// SIMATIC S7-200 project (STEP 7-Micro/WIN), CPU 224XP REL 02.01

SYMBOL_TABLE USUARIO1
S1_VERDE         Q0.0
S1_AMBAR         Q0.1
S1_ROJO          Q0.2
S2_VERDE         Q0.3
S2_AMBAR         Q0.4
S2_ROJO          Q0.5
END_SYMBOL_TABLE

SYMBOL_TABLE Símbolos S7-200
Primer_ciclo_ON  SM0.1    // ON sólo en el primer ciclo
END_SYMBOL_TABLE

ORGANIZATION_BLOCK PRINCIPAL:OB1
TITLE=COMENTARIOS DEL PROGRAMA
BEGIN
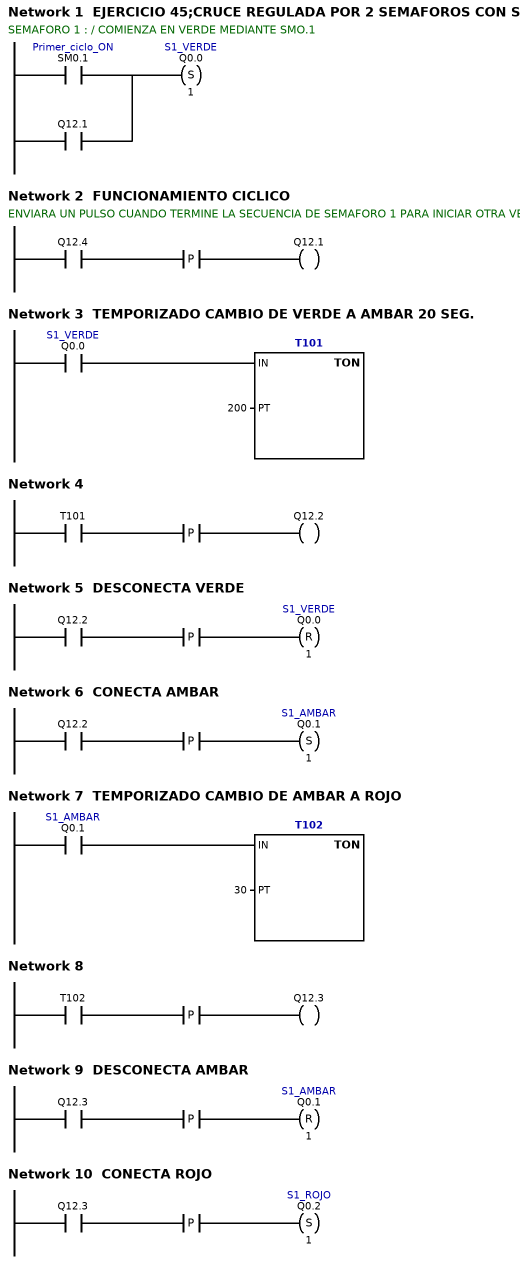
Network 1 // EJERCICIO 45;CRUCE REGULADA POR 2 SEMAFOROS CON SECUENCIA TEMPORIZADAS INDEPENDIENTES.
// SEMAFORO 1 :
// COMIENZA EN VERDE MEDIANTE SMO.1
LD     Primer_ciclo_ON:SM0.1
O      Q12.1
S      S1_VERDE:Q0.0, 1
Network 2 // FUNCIONAMIENTO CICLICO
// ENVIARA UN PULSO CUANDO TERMINE LA SECUENCIA DE SEMAFORO 1 PARA INICIAR OTRA VEZ LA SECUENCIA.
LD     Q12.4
EU
=      Q12.1
Network 3 // TEMPORIZADO CAMBIO DE VERDE A AMBAR 20 SEG.
LD     S1_VERDE:Q0.0
TON    T101, 200
Network 4
LD     T101
EU
=      Q12.2
Network 5 // DESCONECTA VERDE 
LD     Q12.2
EU
R      S1_VERDE:Q0.0, 1
Network 6 // CONECTA AMBAR
LD     Q12.2
EU
S      S1_AMBAR:Q0.1, 1
Network 7 // TEMPORIZADO CAMBIO DE AMBAR A ROJO
LD     S1_AMBAR:Q0.1
TON    T102, 30
Network 8
LD     T102
EU
=      Q12.3
Network 9 // DESCONECTA AMBAR
LD     Q12.3
EU
R      S1_AMBAR:Q0.1, 1
Network 10 // CONECTA ROJO
LD     Q12.3
EU
S      S1_ROJO:Q0.2, 1
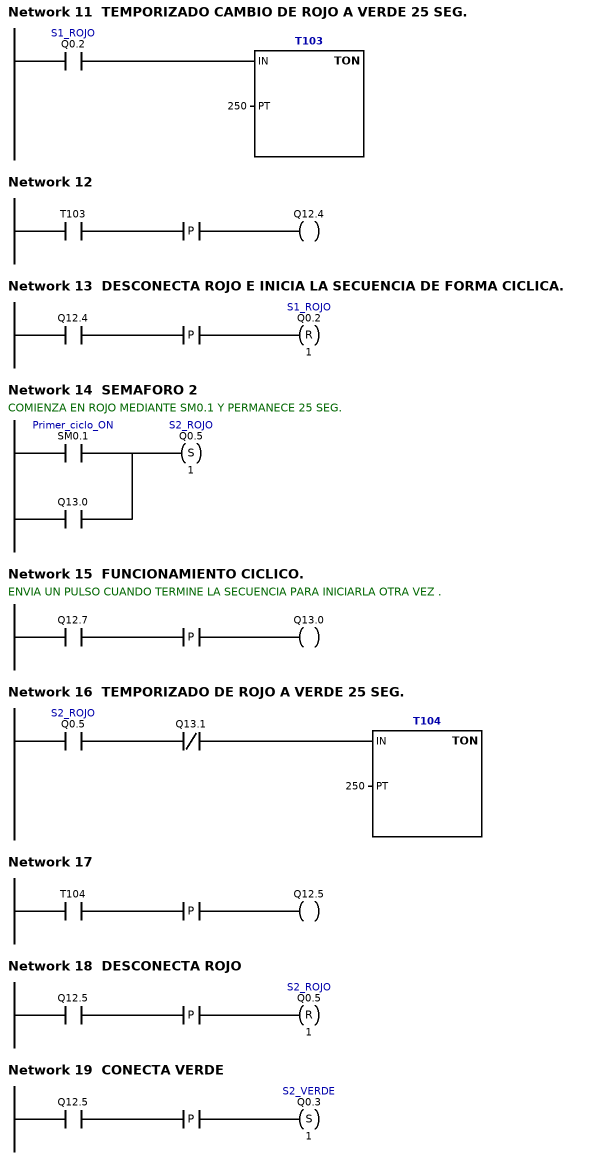
Network 11 // TEMPORIZADO CAMBIO DE ROJO A VERDE 25 SEG.
LD     S1_ROJO:Q0.2
TON    T103, 250
Network 12
LD     T103
EU
=      Q12.4
Network 13 // DESCONECTA ROJO E INICIA LA SECUENCIA DE FORMA CICLICA.
LD     Q12.4
EU
R      S1_ROJO:Q0.2, 1
Network 14 // SEMAFORO 2 
// COMIENZA EN ROJO MEDIANTE SM0.1 Y PERMANECE 25 SEG.
LD     Primer_ciclo_ON:SM0.1
O      Q13.0
S      S2_ROJO:Q0.5, 1
Network 15 // FUNCIONAMIENTO CICLICO.
// ENVIA UN PULSO CUANDO TERMINE LA SECUENCIA PARA INICIARLA OTRA VEZ .
LD     Q12.7
EU
=      Q13.0
Network 16 // TEMPORIZADO DE ROJO A VERDE 25 SEG.
LD     S2_ROJO:Q0.5
AN     Q13.1
TON    T104, 250
Network 17
LD     T104
EU
=      Q12.5
Network 18 // DESCONECTA ROJO
LD     Q12.5
EU
R      S2_ROJO:Q0.5, 1
Network 19 // CONECTA VERDE
LD     Q12.5
EU
S      S2_VERDE:Q0.3, 1
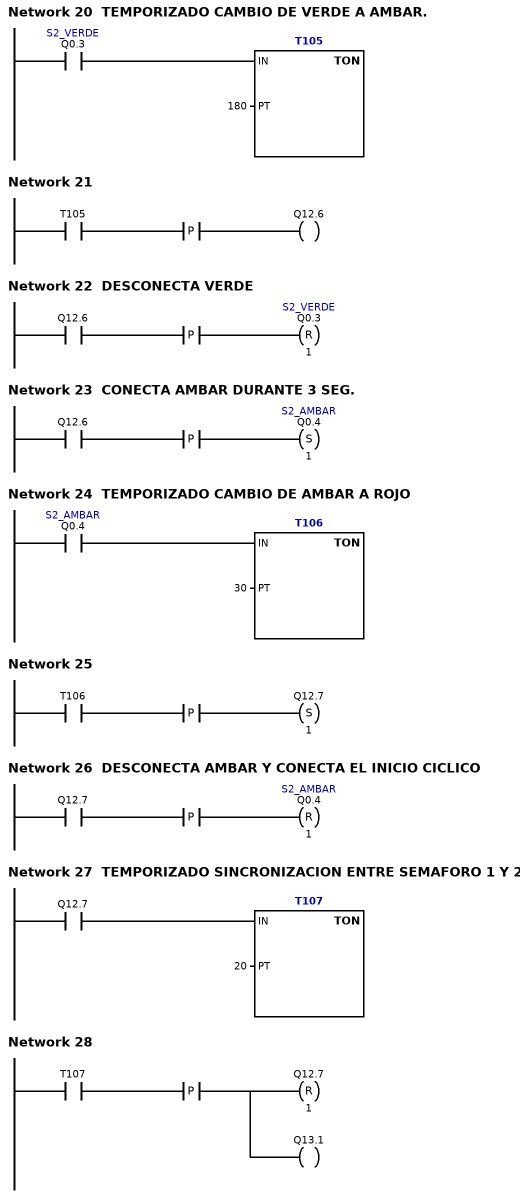
Network 20 // TEMPORIZADO CAMBIO DE VERDE A AMBAR.
LD     S2_VERDE:Q0.3
TON    T105, 180
Network 21
LD     T105
EU
=      Q12.6
Network 22 // DESCONECTA VERDE 
LD     Q12.6
EU
R      S2_VERDE:Q0.3, 1
Network 23 // CONECTA AMBAR DURANTE 3 SEG.
LD     Q12.6
EU
S      S2_AMBAR:Q0.4, 1
Network 24 // TEMPORIZADO CAMBIO DE AMBAR A ROJO
LD     S2_AMBAR:Q0.4
TON    T106, 30
Network 25
LD     T106
EU
S      Q12.7, 1
Network 26 // DESCONECTA AMBAR Y CONECTA EL INICIO CICLICO
LD     Q12.7
EU
R      S2_AMBAR:Q0.4, 1
Network 27 // TEMPORIZADO SINCRONIZACION ENTRE SEMAFORO 1 Y 2 
LD     Q12.7
TON    T107, 20
Network 28
LD     T107
EU
R      Q12.7, 1
=      Q13.1
END_ORGANIZATION_BLOCK
